INTERFACE ITcoState EXTENDS ITcoObject, ITcoRestorable

METHOD ChangeState : ITcoState
VAR_INPUT
	NewState : INT;
END_VAR
END_METHOD

PROPERTY ChangeStateCycle : ULINT
GET
END_GET
END_PROPERTY

PROPERTY EnableAutoRestore : BOOL
GET
END_GET
END_PROPERTY

PROPERTY LastChangedState : INT
GET
END_GET
END_PROPERTY

METHOD OnStateChange
VAR_INPUT
	PreviousState	: INT;
	NewState 		: INT;
END_VAR
END_METHOD

METHOD RestoreObject : ITcoState
VAR_INPUT
	Obj : ITcoRestorable;
END_VAR
END_METHOD

PROPERTY State : INT
GET
END_GET
END_PROPERTY

END_INTERFACE

(* stored: Version 1.1.0.1, ProductVersion 3.1.4024.6
   Itf ITcoState: Id {c649817a-92de-4bd9-bb87-c0d72fad7509}
   Method ChangeState: Id {736c5d1d-d3a0-4eb9-a1f6-eb86c1a20f8f}
   Property ChangeStateCycle: Id {92216c9b-4911-48a2-a6ff-b6246c33da8c}
   Get Get: Id {78ddabb3-69a5-4bb1-a9d6-f1af6af00fdd}
   Property EnableAutoRestore: Id {919401ee-55fe-4554-8ddf-1a407786ef18}
   Get Get: Id {87b763ca-6a82-43eb-8730-8dd9412bbc83}
   Property LastChangedState: Id {d7f49349-dcb2-0003-35b2-44fb772e2dd5}
   Get Get: Id {dbb0a716-7e74-0b51-3177-f946af2212d2}
   Method OnStateChange: Id {93559809-93bd-434a-8b11-9eed96ecef32}
   Method RestoreObject: Id {4a8a2884-a04a-427f-a212-93f7d99ca614}
   Property State: Id {ffa51ee9-dcc1-48dd-ac68-d06a65059caf}
   Get Get: Id {b970a776-b81b-430c-827a-7496827f2909} *)
